FUNCTION_BLOCK CEN_SERVER (* Basic Function Block Type *)
  (* Standard: 61499-2 *)
  (* Version 0.2, 2003-12-04, JHC, Rockwell Automation, Renamed for better indexing. *)
  (* Version 0.1, 2002-11-05, JHC, Rockwell Automation, Corrected missing ST element in Algorithm REQ. *)
  (* Version 0.0, 2000-05-30, JHC, Rockwell Automation *)
  (* Compiler header: package fb.rt.cs725; *)
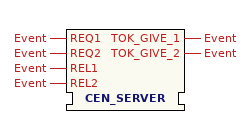
  EVENT_INPUT
    REQ1;
    REQ2;
    REL1;
    REL2;
  END_EVENT
  EVENT_OUTPUT
    TOK_GIVE_1;
    TOK_GIVE_2;
  END_EVENT
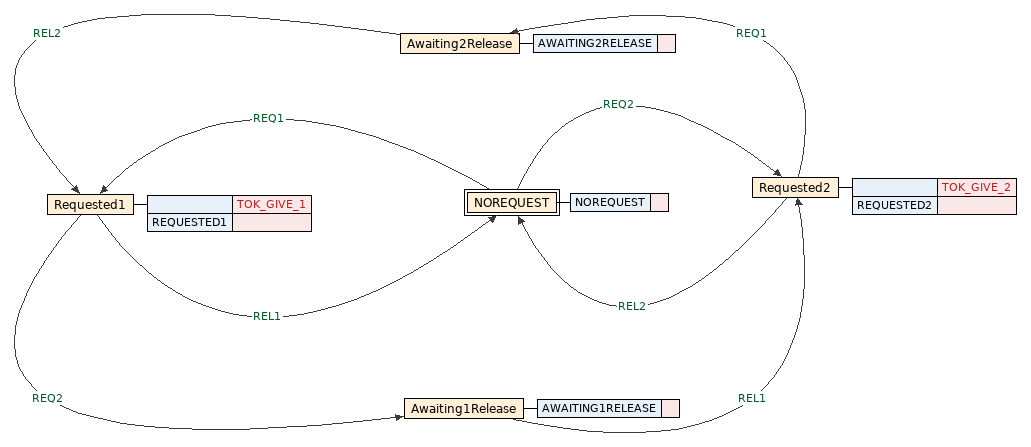
  EC_STATES
    NOREQUEST : NOREQUEST; (* Initial State *)
    Requested1 : -> TOK_GIVE_1, REQUESTED1;
    Requested2 : -> TOK_GIVE_2, REQUESTED2;
    Awaiting1Release : AWAITING1RELEASE;
    Awaiting2Release : AWAITING2RELEASE;
  END_STATES
  EC_TRANSITIONS
    NOREQUEST TO Requested2 := REQ2;
    NOREQUEST TO Requested1 := REQ1;
    Requested2 TO NOREQUEST := REL2;
    Requested1 TO NOREQUEST := REL1;
    Requested1 TO Awaiting1Release := REQ2;
    Awaiting1Release TO Requested2 := REL1;
    Requested2 TO Awaiting2Release := REQ1;
    Awaiting2Release TO Requested1 := REL2;
  END_TRANSITIONS
  ALGORITHM NOREQUEST IN Java:
System.out.println("Server: NOREQUEST");
  END_ALGORITHM
  ALGORITHM REQUESTED2 IN Java:
System.out.println("Server: REQUESTED2");
  END_ALGORITHM
  ALGORITHM REQUESTED1 IN Java:
System.out.println("Server: REQUESTED1");
  END_ALGORITHM
  ALGORITHM AWAITING1RELEASE IN Java:
System.out.println("Server: AWAITING1RELEASE");
  END_ALGORITHM
  ALGORITHM AWAITING2RELEASE IN Java:
System.out.println("Server: AWAITING2RELEASE");
  END_ALGORITHM
END_FUNCTION_BLOCK
